TYPE ST_CommunicationConfig_1 :
STRUCT

    sIpAddress : STRING(15) := '192.168.0.10';
    nPort : UINT := 7171;
	sUsername: STRING(128):= '';
    sPassword : STRING(128) := '';
    tTimeout : TIME := T#5S;
    bAutoReconnect : BOOL := TRUE;
END_STRUCT
END_TYPE

(* stored: Version 1.1.0.1, ProductVersion 3.1.4026.18
   DUT ST_CommunicationConfig_1: Id {949d2472-c6bf-49f3-aeb3-8e259f190a96} *)
